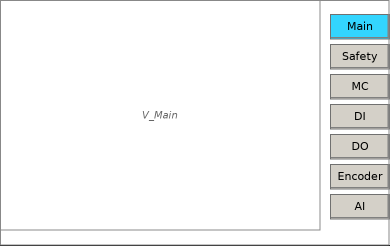
VISUALIZATION V_MainScreen  // 390x246
    Button (330,14 60x25), "Main", input disabled if: HMI_IO.HMI_Page = 1
        OnMouseClick: FrameSelectionChange Selection=SelectedFrame=ca35193f-53d6-45b7-b8b5-0860b53cf110, GlobSel=AssignType=Directly, SelType=Locally
        OnMouseClick: execute { HMI_IO.HMI_Page := 1; }
    Button (330,44 60x25), "Safety", input disabled if: HMI_IO.HMI_Page = 2
        OnMouseClick: FrameSelectionChange Selection=SelectedFrame=ca35193f-53d6-45b7-b8b5-0860b53cf110, Selection=1, GlobSel=AssignType=Directly, SelType=Locally
        OnMouseClick: execute { HMI_IO.HMI_Page := 2; }
    Button (330,74 60x25), "MC", input disabled if: HMI_IO.HMI_Page = 3
        OnMouseClick: FrameSelectionChange Selection=SelectedFrame=ca35193f-53d6-45b7-b8b5-0860b53cf110, Selection=2, GlobSel=AssignType=Directly, SelType=Locally
        OnMouseClick: execute { HMI_IO.HMI_Page := 3; }
    Button (330,104 60x25), "DI", input disabled if: HMI_IO.HMI_Page = 4
        OnMouseClick: FrameSelectionChange Selection=SelectedFrame=ca35193f-53d6-45b7-b8b5-0860b53cf110, Selection=3, GlobSel=AssignType=Directly, SelType=Locally
        OnMouseClick: execute { HMI_IO.HMI_Page := 4; }
    Button (330,134 60x25), "DO", input disabled if: HMI_IO.HMI_Page = 5
        OnMouseClick: FrameSelectionChange Selection=SelectedFrame=ca35193f-53d6-45b7-b8b5-0860b53cf110, Selection=4, GlobSel=AssignType=Directly, SelType=Locally
        OnMouseClick: execute { HMI_IO.HMI_Page := 5; }
    Button (330,164 60x25), "Encoder", input disabled if: HMI_IO.HMI_Page = 6
        OnMouseClick: FrameSelectionChange Selection=SelectedFrame=ca35193f-53d6-45b7-b8b5-0860b53cf110, Selection=5, GlobSel=AssignType=Directly, SelType=Locally
        OnMouseClick: execute { HMI_IO.HMI_Page := 6; }
    Button (330,194 60x25), "AI", input disabled if: HMI_IO.HMI_Page = 7
        OnMouseClick: FrameSelectionChange Selection=SelectedFrame=ca35193f-53d6-45b7-b8b5-0860b53cf110, Selection=6, GlobSel=AssignType=Directly, SelType=Locally
        OnMouseClick: execute { HMI_IO.HMI_Page := 7; }
    Line (0,245) (390,245)
    Frame (0,0 320x230)
        shows V_Main()
        shows V_Safety()
        shows V_MC()
        shows V_DI()
        shows V_DO()
        shows V_Encoder()
        shows V_AI()
END_VISUALIZATION

(* stored: Version 1.1.0.1, ProductVersion 3.1.4024.11
   Visu V_MainScreen: Id {a6aa1a41-be82-422d-9649-bd282432e6d5} *)
